PROGRAM MAIN
VAR
	iSelection : INT := 1;

END_VAR


CASE iSelection OF
	
	1:
	gameMode301();

	
END_CASE

END_PROGRAM

(* stored: Version 1.1.0.1, ProductVersion 3.1.4024.12
   POU MAIN: Id {40a5c440-309e-4fa5-8cc4-c4f078c698bd}, SpecialFunc None *)
